(* CODESYS project SortingByHeight_Basic.project

Project tree, tasks and I/O mapping:
  Device : CODESYS Control Win V3, 3S - Smart Software Solutions GmbH, order no. 305021, version 3.5.11.30
    application Application
      libraries: Standard, * (System)
      task MainTask (cyclic, interval t#20ms, priority 1) calls PLC_PRG
      program PLC_PRG [LD]
      global variables GVL
      Symbols
*)

// Device/Application/GVL
{attribute 'qualified_only'}
VAR_GLOBAL
	p1: BOOL;
	t1: BOOL;
	start: BOOL;
	p2: BOOL;
	palletSensor: BOOL;
	t2: BOOL;
	p3: BOOL;
	t3: BOOL;
	p4: BOOL;
	loaded: BOOL;
	t4: BOOL;
	p5: BOOL;
	alto: BOOL;
	t5: BOOL;
	p6: BOOL;
	atLeftEntry: BOOL;
	t6: BOOL;
	p7: BOOL;
	atLeftExit: BOOL;
	t7: BOOL;
	p8: BOOL;
	t8: BOOL;
	t9: BOOL;
	atRightEntry: BOOL;
	p9: BOOL;
	atRightExit: BOOL;
	t10: BOOL;
	p10: BOOL;
	t11: BOOL;
	p11: BOOL;
	stop: BOOL;
	t12: BOOL;
	p12: BOOL;
	t13: BOOL;
	reset: BOOL;
	t14: BOOL;
	p13: BOOL;
	t15: BOOL;
	p14: BOOL;
	t16: BOOL;
	highSensor: BOOL;
	p15: BOOL;
	t17: BOOL;
	p16: BOOL;
	aux0: BOOL;
	CTU_0: CTU;
	contador: INT;
	conveyorEntry: BOOL;
	load: BOOL;
	transferLeft: BOOL;
	transferRight: BOOL;
	conveyorLeft: BOOL;
	conveyorRight: BOOL;
END_VAR

// Device/Application/PLC_PRG
PROGRAM PLC_PRG
VAR
	p1: BOOL;
	t1: BOOL;
	start: BOOL;
	p2: BOOL;
	palletSensor: BOOL;
	t2: BOOL;
	p3: BOOL;
	t3: BOOL;
	p4: BOOL;
	loaded: BOOL;
	t4: BOOL;
	p5: BOOL;
	alto: BOOL;
	t5: BOOL;
	p6: BOOL;
	atLeftEntry: BOOL;
	t6: BOOL;
	p7: BOOL;
	atLeftExit: BOOL;
	t7: BOOL;
	p8: BOOL;
	t8: BOOL;
	t9: BOOL;
	atRightEntry: BOOL;
	p9: BOOL;
	atRightExit: BOOL;
	t10: BOOL;
	p10: BOOL;
	t11: BOOL;
	p11: BOOL;
	stop: BOOL;
	t12: BOOL;
	p12: BOOL;
	t13: BOOL;
	reset: BOOL;
	t14: BOOL;
	p13: BOOL;
	t15: BOOL;
	p14: BOOL;
	t16: BOOL;
	highSensor: BOOL;
	p15: BOOL;
	t17: BOOL;
	p16: BOOL;
	aux0: BOOL;
	CTU_0: CTU;
	contador: INT;
	conveyorEntry: BOOL;
	load: BOOL;
	transferLeft: BOOL;
	transferRight: BOOL;
	conveyorLeft: BOOL;
	conveyorRight: BOOL;
	desligar: BOOL;
END_VAR
VAR // added by the converter: edge detectors and wires of the graphical bodies
    _rt1, _rt2, _rt3, _rt4, _rt5, _rt6 : R_TRIG;
    _w1, _w2, _w3 : BOOL;
END_VAR

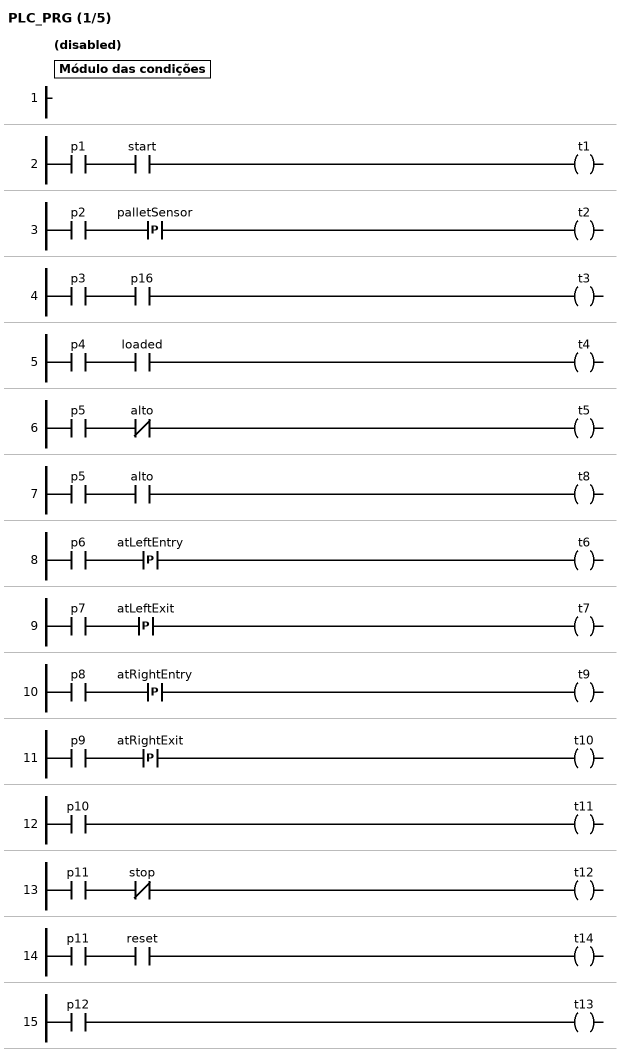
// NETWORK 1 (disabled)
// label: Módulo das condições

// NETWORK 2
t1 := p1 AND start;

// NETWORK 3
_rt1(CLK := palletSensor);
t2 := p2 AND _rt1.Q;

// NETWORK 4
t3 := p3 AND p16;

// NETWORK 5
t4 := p4 AND loaded;

// NETWORK 6
t5 := p5 AND NOT alto;

// NETWORK 7
t8 := p5 AND alto;

// NETWORK 8
_rt2(CLK := atLeftEntry);
t6 := p6 AND _rt2.Q;

// NETWORK 9
_rt3(CLK := atLeftExit);
t7 := p7 AND _rt3.Q;

// NETWORK 10
_rt4(CLK := atRightEntry);
t9 := p8 AND _rt4.Q;

// NETWORK 11
_rt5(CLK := atRightExit);
t10 := p9 AND _rt5.Q;

// NETWORK 12
t11 := p10;

// NETWORK 13
t12 := p11 AND NOT stop;

// NETWORK 14
t14 := p11 AND reset;

// NETWORK 15
t13 := p12;

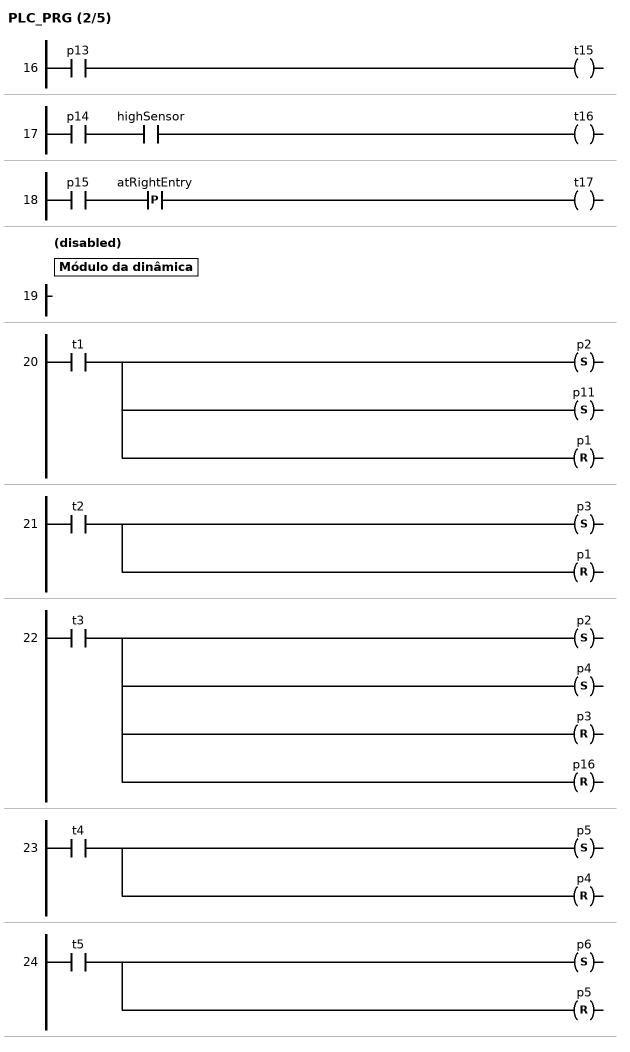
// NETWORK 16
t15 := p13;

// NETWORK 17
t16 := p14 AND highSensor;

// NETWORK 18
_rt6(CLK := atRightEntry);
t17 := p15 AND _rt6.Q;

// NETWORK 19 (disabled)
// label: Módulo da dinâmica

// NETWORK 20
p2 S= t1;
p11 S= t1;
p1 R= t1;

// NETWORK 21
p3 S= t2;
p1 R= t2;

// NETWORK 22
p2 S= t3;
p4 S= t3;
p3 R= t3;
p16 R= t3;

// NETWORK 23
p5 S= t4;
p4 R= t4;

// NETWORK 24
p6 S= t5;
p5 R= t5;

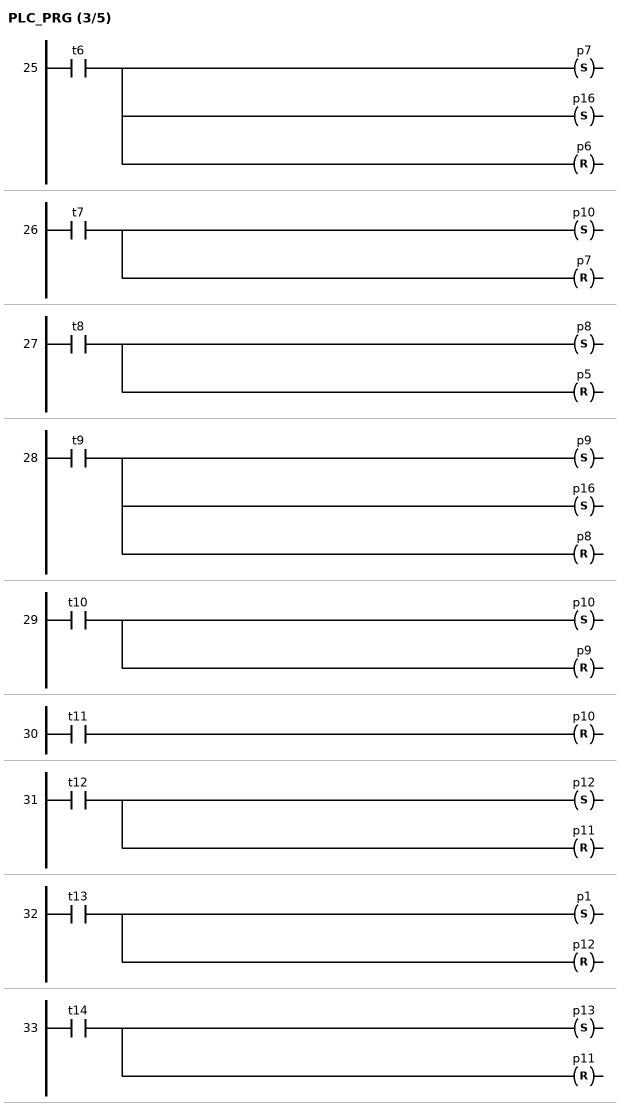
// NETWORK 25
p7 S= t6;
p16 S= t6;
p6 R= t6;

// NETWORK 26
p10 S= t7;
p7 R= t7;

// NETWORK 27
p8 S= t8;
p5 R= t8;

// NETWORK 28
p9 S= t9;
p16 S= t9;
p8 R= t9;

// NETWORK 29
p10 S= t10;
p9 R= t10;

// NETWORK 30
p10 R= t11;

// NETWORK 31
p12 S= t12;
p11 R= t12;

// NETWORK 32
p1 S= t13;
p12 R= t13;

// NETWORK 33
p13 S= t14;
p11 R= t14;

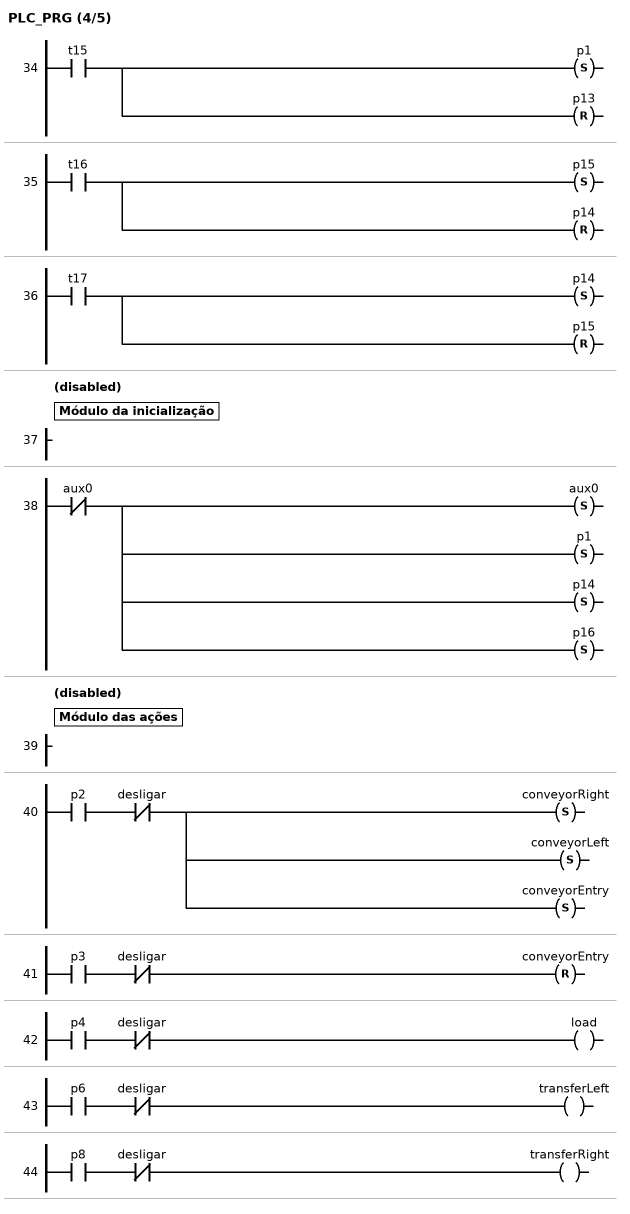
// NETWORK 34
p1 S= t15;
p13 R= t15;

// NETWORK 35
p15 S= t16;
p14 R= t16;

// NETWORK 36
p14 S= t17;
p15 R= t17;

// NETWORK 37 (disabled)
// label: Módulo da inicialização

// NETWORK 38
_w1 := NOT aux0;
aux0 S= _w1;
p1 S= _w1;
p14 S= _w1;
p16 S= _w1;

// NETWORK 39 (disabled)
// label: Módulo das ações

// NETWORK 40
_w2 := p2 AND NOT desligar;
conveyorRight S= _w2;
conveyorLeft S= _w2;
conveyorEntry S= _w2;

// NETWORK 41
conveyorEntry R= p3 AND NOT desligar;

// NETWORK 42
load := p4 AND NOT desligar;

// NETWORK 43
transferLeft := p6 AND NOT desligar;

// NETWORK 44
transferRight := p8 AND NOT desligar;

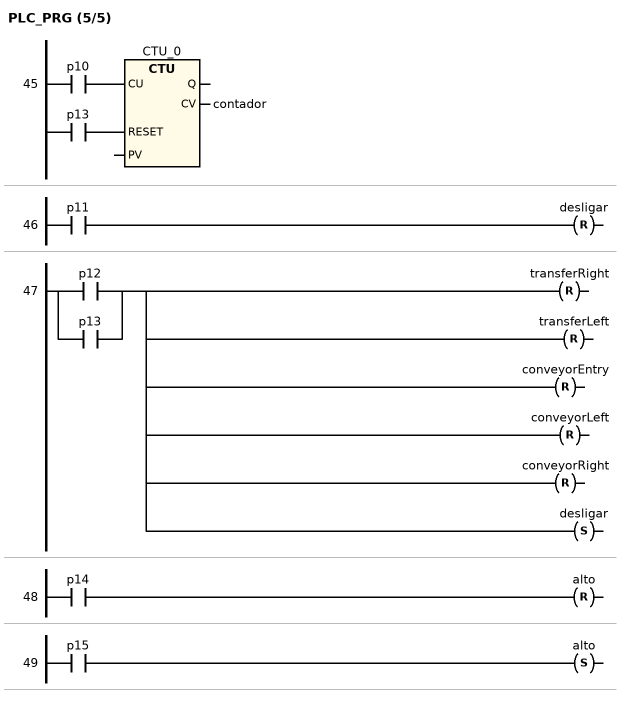
// NETWORK 45
CTU_0(CU := p10, RESET := p13, CV => contador); // CTU

// NETWORK 46
desligar R= p11;

// NETWORK 47
_w3 := p12 OR p13;
transferRight R= _w3;
transferLeft R= _w3;
conveyorEntry R= _w3;
conveyorLeft R= _w3;
conveyorRight R= _w3;
desligar S= _w3;

// NETWORK 48
alto R= p14;

// NETWORK 49
alto S= p15;

END_PROGRAM
